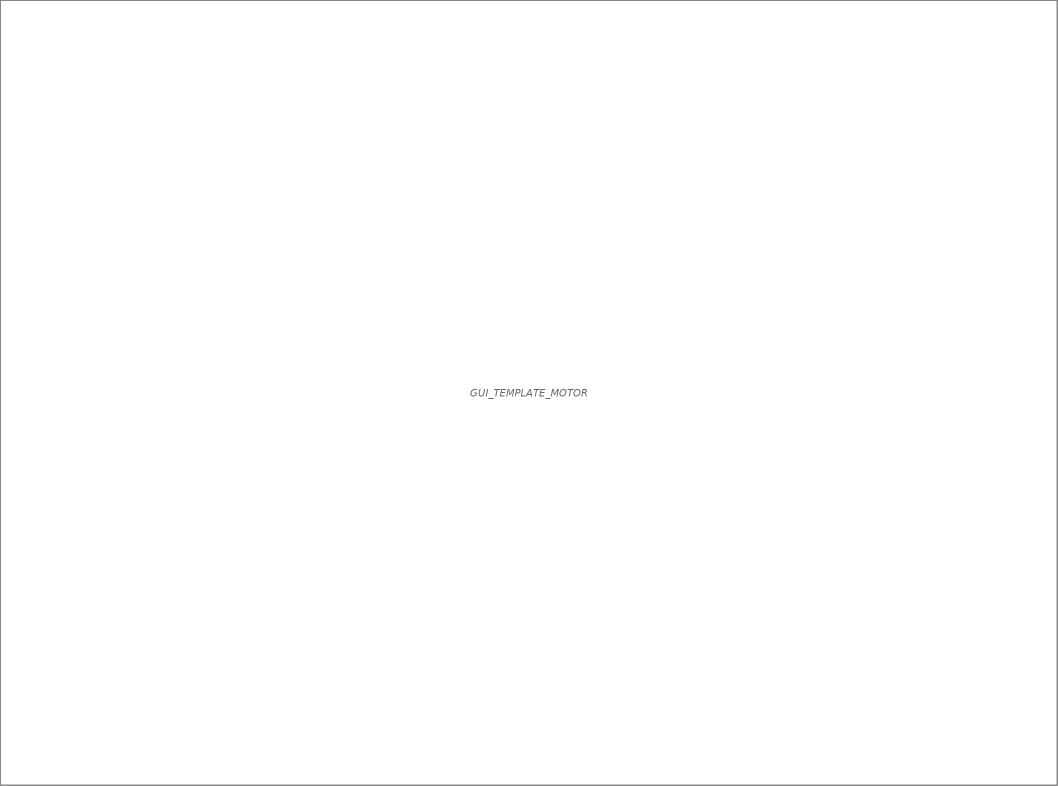
VISUALIZATION GUI_NOTT_NBS  // 1058x786
    Frame (0,0 1058x786)
        shows GUI_TEMPLATE_MOTOR(m_Instance := MAIN.nott_ics.Calibration_Unit_Beam_Splitter.NBS)
END_VISUALIZATION

(* stored: Version 1.1.0.1, ProductVersion 3.1.4024.14
   Visu GUI_NOTT_NBS: Id {5443c129-ab2e-4c2c-a3de-6ad6b0d3f786} *)
